// TIA Portal V16 export
// export: Created 2023-03-29T11:03:36.5859649Z, ExportSetting WithDefaults, DisplayName Totally Integrated Automation Portal, DisplayVersion V16 Update 6, DisplayName TIA Portal Version Control Interface, DisplayVersion V16 Update 2, DisplayName TIA Portal Openness, DisplayVersion V16 Update 6, DisplayName STEP 7 Professional, DisplayVersion V16 Update 6, DisplayName STEP 7 Safety, DisplayVersion V16, DisplayName WinCC Advanced, DisplayVersion V16 Update 6
DATA_BLOCK "EX012_ErrorBuffer_OB82"   // DB103
TITLE = BufferOB82
{ S7_Optimized_Access := 'TRUE' }
AUTHOR : Gilewski
VERSION : 0.1
// Data block for OB82 buffer
// stored: AutoNumber false, DBAccessibleFromOPCUA true, IsOnlyStoredInLoadMemory false, IsRetainMemResEnabled false, IsWriteProtectedInAS false, MemoryReserve 100
   VAR RETAIN
      OB82ErrorCounter : USInt;   // //Counter for error buffer
      CounterDiagStatusUpdate : USInt;   // //Counter for another error
      ErrorDataOB82 { S7_SetPoint := 'True'} : Array[1..200] of "stt_OB82";   // //buffer for error from OB82
   END_VAR
BEGIN
END_DATA_BLOCK
